# EPICS substitutions: vacuum/MAIN_TRUNK/vacApp/Db/bc3s_agilent4uhv.substitutions
# Agilent4UHV substitutions file

file db/agilent4uhv.db
{
     pattern {LOCA,			DEV,		PORT,		ADDR,	TIMEOUT}
     		 {SL3,			BC3S,		4uhv_1,		0,		0.2}
}
file db/agilent4uhv_alias.db
{
     pattern {LOCA,			DEV,		SUB1,					SUB2,					SUB3,						SUB4,				PORT,	ADDR,	TIMEOUT}
     		 {SL3,			BC3S,	IP01,		IP02,		IP03,			IP04,	4uhv_1,	0,		0.2}
}
